FUNCTION_BLOCK DataPanel_xDB_16_PWM_SAE_J1939 (* Service Interface Function Block Type *)
  (* Standard: SAE J1939; Function: All Outputs: Unpaired PWM/PWM(i); Type: DP-34044-3-000; Description: this maps to QX *)
  (* Version 1.0, 2018-12-05, Jose Cabral *)
  (* Version 1.1, 2022-08-04, Franz Höpfinger, HR Agrartechnik GmbH *)
  (* Version 1.2, 2023-01-05, Franz Höpfinger, HR Agrartechnik GmbH *)
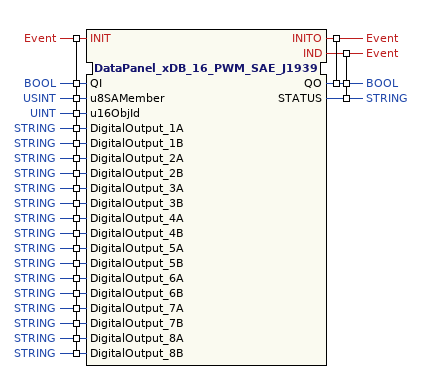
  EVENT_INPUT
    INIT WITH QI, u8SAMember, u16ObjId, DigitalOutput_1A, DigitalOutput_1B, DigitalOutput_2A, DigitalOutput_2B, DigitalOutput_3A, DigitalOutput_3B, DigitalOutput_4A, DigitalOutput_4B, DigitalOutput_5A, DigitalOutput_5B, DigitalOutput_6A, DigitalOutput_6B, DigitalOutput_7A, DigitalOutput_7B, DigitalOutput_8A, DigitalOutput_8B; (* Service Initialization *)
  END_EVENT
  EVENT_OUTPUT
    INITO WITH QO; (* Initialization Confirm *)
    IND WITH QO, STATUS; (* Indication from Resource *)
  END_EVENT
  VAR_INPUT
    QI : BOOL; (* Event Input Qualifier *)
    u8SAMember : USINT := 224; (* Node SA 224..239 *)
    u16ObjId : UINT := 65535; (* Dummy ! set to 65535 if in Doubt. 0 deactivates FB. *)
    DigitalOutput_1A : STRING;
    DigitalOutput_1B : STRING;
    DigitalOutput_2A : STRING;
    DigitalOutput_2B : STRING;
    DigitalOutput_3A : STRING;
    DigitalOutput_3B : STRING;
    DigitalOutput_4A : STRING;
    DigitalOutput_4B : STRING;
    DigitalOutput_5A : STRING;
    DigitalOutput_5B : STRING;
    DigitalOutput_6A : STRING;
    DigitalOutput_6B : STRING;
    DigitalOutput_7A : STRING;
    DigitalOutput_7B : STRING;
    DigitalOutput_8A : STRING;
    DigitalOutput_8B : STRING;
  END_VAR
  VAR_OUTPUT
    QO : BOOL; (* Event Output Qualifier *)
    STATUS : STRING; (* Service Status *)
  END_VAR
END_FUNCTION_BLOCK
